FUNCTION SPLIT_WORD_INTO_QUARTERS (* this Function extracts the 8 QUARTER BYTE from a word *)
  (* Standard: 61499-1; Description: Copyright (c) 2024 HR Agrartechnik GmbH This program and the accompanying materials are made available under the terms of the Eclipse Public License 2.0 which is available at https://www.eclipse.org/legal/epl-2.0/ SPDX-License-Identifier: EPL-2.0 *)
  (* Version 3.0.1, 2026-09-29, Martin Jobst, fix ST package declaration *)
  (* Version 3.0, 2025-04-14, Patrick Aigner, changed package *)
  (* Version 1.1, 2024-07-24, Moritz Ortmeier, HR Agrartechnik, rename Function and change Output Variables *)
  (* Version 1.0, 2024-02-22, Franz Höpfinger, HR Agrartechnik, initial Implementation *)
  PACKAGE eclipse4diac::utils::splitting;
  IMPORT eclipse4diac::utils::const::quarterconst;
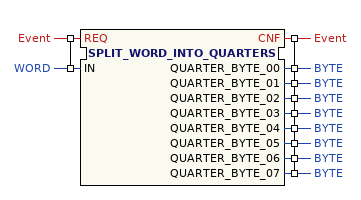
  EVENT_INPUT
    REQ WITH IN;
  END_EVENT
  EVENT_OUTPUT
    CNF WITH QUARTER_BYTE_00, QUARTER_BYTE_01, QUARTER_BYTE_02, QUARTER_BYTE_03, QUARTER_BYTE_04, QUARTER_BYTE_05, QUARTER_BYTE_06, QUARTER_BYTE_07;
  END_EVENT
  VAR_INPUT
    IN : WORD;
  END_VAR
  VAR_OUTPUT
    QUARTER_BYTE_00 : BYTE;
    QUARTER_BYTE_01 : BYTE;
    QUARTER_BYTE_02 : BYTE;
    QUARTER_BYTE_03 : BYTE;
    QUARTER_BYTE_04 : BYTE;
    QUARTER_BYTE_05 : BYTE;
    QUARTER_BYTE_06 : BYTE;
    QUARTER_BYTE_07 : BYTE;
  END_VAR
  BODY IN ST:
PACKAGE eclipse4diac::utils::splitting;

IMPORT eclipse4diac::utils::const::quarterconst;

(* this Function extracts the 8 QUARTER BYTE from a word *)
FUNCTION SPLIT_WORD_INTO_QUARTERS

VAR_INPUT
	IN : WORD;
END_VAR

VAR_OUTPUT
	QUARTER_BYTE_00 : BYTE;
	QUARTER_BYTE_01 : BYTE;
	QUARTER_BYTE_02 : BYTE;
	QUARTER_BYTE_03 : BYTE;
	QUARTER_BYTE_04 : BYTE;
	QUARTER_BYTE_05 : BYTE;
	QUARTER_BYTE_06 : BYTE;
	QUARTER_BYTE_07 : BYTE;
END_VAR

QUARTER_BYTE_00 := WORD_TO_BYTE(SHR(IN AND quarterconst::WORD_QUARTER_00, quarterconst::SHIFT_QUARTER_00));
QUARTER_BYTE_01 := WORD_TO_BYTE(SHR(IN AND quarterconst::WORD_QUARTER_01, quarterconst::SHIFT_QUARTER_01));
QUARTER_BYTE_02 := WORD_TO_BYTE(SHR(IN AND quarterconst::WORD_QUARTER_02, quarterconst::SHIFT_QUARTER_02));
QUARTER_BYTE_03 := WORD_TO_BYTE(SHR(IN AND quarterconst::WORD_QUARTER_03, quarterconst::SHIFT_QUARTER_03));
QUARTER_BYTE_04 := WORD_TO_BYTE(SHR(IN AND quarterconst::WORD_QUARTER_04, quarterconst::SHIFT_QUARTER_04));
QUARTER_BYTE_05 := WORD_TO_BYTE(SHR(IN AND quarterconst::WORD_QUARTER_05, quarterconst::SHIFT_QUARTER_05));
QUARTER_BYTE_06 := WORD_TO_BYTE(SHR(IN AND quarterconst::WORD_QUARTER_06, quarterconst::SHIFT_QUARTER_06));
QUARTER_BYTE_07 := WORD_TO_BYTE(SHR(IN AND quarterconst::WORD_QUARTER_07, quarterconst::SHIFT_QUARTER_07));

END_FUNCTION
  END_BODY
END_FUNCTION
